// TIA Portal V19 export
TYPE "Decoiler_Status"
   STRUCT
      Feed : "SpeedMachine_COut";
      Jaws : "ValveMachine_COut";
      Coupling : "ValveMachine_COut";
      SnubberLift : "ValveMachine_COut";
      SnubberRoll : "ValveMachine_COut";
      CoilDiameter { S7_SetPoint := 'True'} : Real;
      EndOfCoil : Bool;
      CouplingEngaged : Bool;
   END_STRUCT;
END_TYPE
